FUNCTION_BLOCK Test_function_block
VAR_INPUT
END_VAR
VAR_OUTPUT
END_VAR
VAR
END_VAR

END_FUNCTION_BLOCK

(* stored: Version 1.1.0.1, ProductVersion 3.1.4024.12
   POU Test_function_block: Id {db30877d-2af4-4c9c-b052-06e3294a70a7}, SpecialFunc None *)
